FUNCTION_BLOCK PAEActValve2 EXTENDS PAEActuator2way
VAR_INPUT
END_VAR
VAR_OUTPUT
END_VAR
VAR
END_VAR

METHOD PUBLIC PAEActValve2
VAR_INPUT
END_VAR
END_METHOD

END_FUNCTION_BLOCK

(* stored: Version 1.1.0.1, ProductVersion 3.1.4020.12
   POU PAEActValve2: Id {a5dc4379-4d48-4d10-b166-f1f4a85e11fd}, SpecialFunc None
   Method PAEActValve2: Id {40871f23-1e77-4e99-9259-9b6a7eb6f729} *)
